// TIA Portal V15.1 export
// export: Created 2024-06-21T08:40:54.2750484Z, ExportSetting WithDefaults, DisplayName Totally Integrated Automation Portal, DisplayVersion V15.1 Update 5, DisplayName TIA Portal Openness, DisplayVersion V15.1 Update 5, DisplayName SINAMICS Startdrive Advanced, DisplayVersion V15.1, DisplayName G130, G150, S120, S150, SINAMICS MV, S210, DisplayVersion V15.1, DisplayName G110M, G120, G120C, G120D, G120P, DisplayVersion V15.1, DisplayName STEP 7 Professional, DisplayVersion V15.1 Update 5, DisplayName STEP 7 Safety, DisplayVersion V15.1, DisplayName WinCC Professional, DisplayVersion V15.1 Update 5, DisplayName SIMATIC Visualization Architect, DisplayVersion V15.1
FUNCTION "LAlarmSummary" : Void   // FC2534, FBD
TITLE = LAlarmSummary
{ S7_Optimized_Access := 'TRUE' }
VERSION : 0.1
// =============================================================================
// This module is used to sum all alarm's from all objects "FB&FC's" and the send it to LMode & LSystemVar-S71500
// =============================================================================
// stored: AutoNumber false, IsIECCheckEnabled false, SetENOAutomatically False, UDAEnableTagReadback false
   VAR_INPUT
      I_AlarmA : Bool;
      I_AlarmB : Bool;   // Alarm B Active in the Modezone
      I_AlarmC : Bool;   // Alarm C Active in the Modezone
      I_AlarmD : Bool;   // Alarm D Active in the Modezone
      I_AlarmABCondition : Bool;   // Alarm AB Condition
   END_VAR
   VAR_IN_OUT
      IO_Alarm : "Alarm";
      C_UpperLevelHW : Bool;   // Configuration Type
      C_UpperLevelSafety : Bool;   // Configuration Type
      C_Safety : Bool;   // Configuration Type
      C_Mechanic : Bool;   // Configuration Type
      C_Transport : Bool;   // Configuration Type
      C_Feature1 : Bool;   // Configuration Type
      C_Feature2 : Bool;   // Configuration Type
      C_Feature3 : Bool;   // Configuration Type
   END_VAR
BEGIN

NETWORK
TITLE = **** 2.2 - Alarms - Alarm generation **** Alarm's Active
// Alarm's Active
// Activate Alarm A
      A     #I_AlarmA;
      S     #IO_Alarm.AlarmAActive;
// Activate Alarm B
      A     #I_AlarmB;
      S     #IO_Alarm.AlarmBActive;

// Activate Alarm C
      A     #I_AlarmC;
      S     #IO_Alarm.AlarmCActive;

// Activate Alarm D
      A     #I_AlarmD;
      S     #IO_Alarm.AlarmDActive;

// Activate AlarmABCondition
      A     #I_AlarmABCondition;
      S     #IO_Alarm.AlarmABCondition;

// Activate Object Not Ok
      A     #C_Mechanic;
      A(;
      O     #I_AlarmA;
      O     #I_AlarmB;
      O     #I_AlarmC;
      );
      S     #IO_Alarm.EnableAlarmMechanicNOk;

// Activate Object Not Ok
      A     #C_Transport;
      A(;
      O     #I_AlarmA;
      O     #I_AlarmB;
      O     #I_AlarmC;
      );
      S     #IO_Alarm.EnableAlarmTransportNOk;


// Activate Object Not Ok
      A     #C_Safety;
      A(;
      O     #I_AlarmA;
      O     #I_AlarmB;
      );
      S     #IO_Alarm.SafetyNok;

// Activate Object Not Ok
      A     #C_UpperLevelSafety;
      A(;
      O     #I_AlarmA;
      O     #I_AlarmB;
      );
      S     #IO_Alarm.SafetyNotOkUpperLevel;

// Activate Object Not Ok
      A     #C_UpperLevelHW;
      A(;
      O     #I_AlarmA;
      O     #I_AlarmB;
      );
      S     #IO_Alarm.UpperLevelHWNok;

// Activate Object Not Ok
      A     #C_Feature1;
      A(;
      O     #I_AlarmA;
      O     #I_AlarmB;
      O     #I_AlarmC;
      );
      S     #IO_Alarm.Feature1;

// Activate Object Not Ok
      A     #C_Feature2;
      A(;
      O     #I_AlarmA;
      O     #I_AlarmB;
      O     #I_AlarmC;
      );
      S     #IO_Alarm.Feature2;

// Activate Object Not Ok
      A     #C_Feature3;
      A(;
      O     #I_AlarmA;
      O     #I_AlarmB;
      O     #I_AlarmC;
      );
      S     #IO_Alarm.Feature3;


END_FUNCTION
